(* Schneider Machine Expert - Basic project proj1_schneider, file version 2.7.0.0 *)
(* ProjectInformations: Name=New project *)

HARDWARE
  Cpu 0: TM221CE40R
  ModuleExtensionObject 0: TM3AQ2/G
  EthernetConfiguration: NetworkName=M221, IpAllocationMode=FixedAddress, IpAddress=0.0.0.0, SubnetMask=0.0.0.0
  SerialLineConfiguration: Baud=Baud19200, Parity=ParityEven, DataBits=DataBits8, StopBits=StopBits1, PhysicalMedium=PhysicalMediumRs485, TransmissionMode=TransmissionModeModbusRtu, SlaveId=1, Addressing=SlaveAddressing
  MastTask: UsePeriodScanMode=false, PeriodScan=100
  FastTask: Period=255
  CpuBehavior: StartingMode=StartAsPreviousState, AutoSaveRamOnEeprom=true, WatchdogPeriod=250

SYMBOLS  (address, symbol, comment, settings)
  %M0       TIMER2
  %M1       TIMER1
  %X1       STEP0
  %X2       STEP1
  %X3       STEP2
  %X4       STEP3
  %TM0        [Preset=1, Base=OneSecond]
  %TM3        [Preset=3, Base=OneSecond]
  %I0.0     BTNSTART
  %I0.20    SENSIND
  %Q0.0     LED
  %Q0.11    BELT_ON
  %Q0.12    ELMAG_ON

GRAFCET Grafcet POU
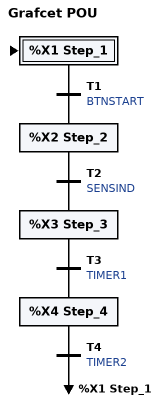
  INITIAL_STEP %X1  (* Step_1 *)
  STEP %X2  (* Step_2 *)
  STEP %X3  (* Step_3 *)
  STEP %X4  (* Step_4 *)
  TRANSITION T1 FROM %X1 TO %X2 := BTNSTART;
  TRANSITION T2 FROM %X2 TO %X3 := SENSIND;
  TRANSITION T3 FROM %X3 TO %X4 := TIMER1;
  TRANSITION T4 FROM %X4 TO %X1 := TIMER2;

POU New POU
  (* SectionNumber=1 *)

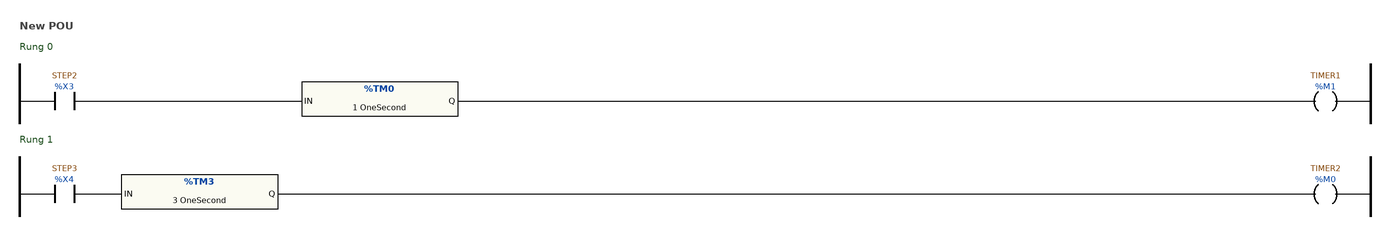

// Rung 0
  BLK %TM0
  LD %X3                  (* STEP2 *)
  IN
  OUT_BLK
  LD Q
  ST %M1                  (* TIMER1 *)
  END_BLK
  // as ST:
  //   %TM0(IN := STEP2);
  //   TIMER1 := %TM0.Q;

// Rung 1
  BLK %TM3
  LD %X4                  (* STEP3 *)
  IN
  OUT_BLK
  LD Q
  ST %M0                  (* TIMER2 *)
  END_BLK
  // as ST:
  //   %TM3(IN := STEP3);
  //   TIMER2 := %TM3.Q;

TRANSITION T1 (%X1 -> %X2) 
  (* SectionNumber=0 *)

// Rung 2: Tr1
  LD %I0.0                (* BTNSTART *)
  ENDT
  // as ST:
  //   TRANSITION := BTNSTART;

TRANSITION T2 (%X2 -> %X3) 
  (* SectionNumber=0 *)

// Rung 3: Tr2
  LD %I0.20               (* SENSIND *)
  ENDT
  // as ST:
  //   TRANSITION := SENSIND;

TRANSITION T3 (%X3 -> %X4) 
  (* SectionNumber=0 *)

// Rung 4: Tr3
  LD %M1                  (* TIMER1 *)
  ENDT
  // as ST:
  //   TRANSITION := TIMER1;

TRANSITION T4 (%X4 -> %X1) 
  (* SectionNumber=0 *)

// Rung 5: Tr4
  LD %M0                  (* TIMER2 *)
  ENDT
  // as ST:
  //   TRANSITION := TIMER2;

POU New POU
  (* SectionNumber=5 *)

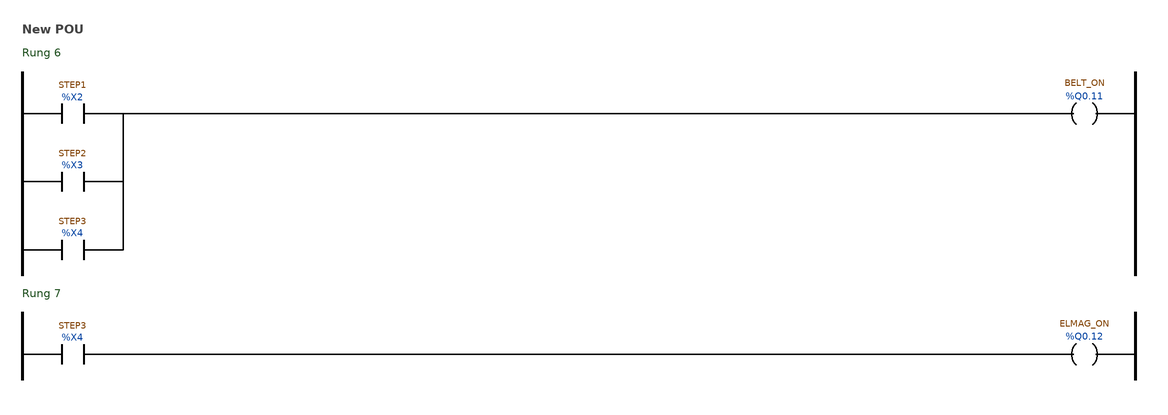

// Rung 6
  LD %X2                  (* STEP1 *)
  OR %X3                  (* STEP2 *)
  OR %X4                  (* STEP3 *)
  ST %Q0.11               (* BELT_ON *)
  // as ST:
  //   BELT_ON := STEP1 OR STEP2 OR STEP3;

// Rung 7
  LD %X4                  (* STEP3 *)
  ST %Q0.12               (* ELMAG_ON *)
  // as ST:
  //   ELMAG_ON := STEP3;
